PROGRAM MAIN
VAR
	b1		:BOOL;
	i1		:INT;
	i2		:INT;
	
	fbADSRead	:ADSREAD;
	fbREdge		:R_TRIG;
	
	bStart		AT %I* :BOOL;
	
END_VAR

FOR i1 := 1 TO 10 BY 1 DO;
	i2:=i2 + 1;
END_FOR

fbADSRead.NETID := '192.168.15.15.1.1';
fbADSRead.PORT := 10500;
fbADSRead.IDXGRP  := 16#2000;
fbADSRead.IDXOFFS := 0;

fbREdge(CLK:=bStart,Q=>);

fbADSRead(
		READ:=fbREdge.Q
		);

END_PROGRAM

(* stored: Version 1.1.0.1, ProductVersion 3.1.4026.8
   POU MAIN: Id {798194bd-2eb4-4ecb-9a48-b0ecad4b7fc9}, SpecialFunc None *)
